MoveJ RelTool (starting_position, 116, -300, -124 \Rx:=7.8, \Ry:=-3, \Rz:=0), v200, z200, Tooldata_7;
MoveJ RelTool (starting_position, 117, -300, -124 \Rx:=7.6, \Ry:=-3, \Rz:=0), v200, z200, Tooldata_7;
MoveJ RelTool (starting_position, 117, -300, -124 \Rx:=7.4, \Ry:=-3, \Rz:=0), v200, z200, Tooldata_7;
MoveJ RelTool (starting_position, 117, -300, -123 \Rx:=7.2, \Ry:=-3, \Rz:=0), v200, z200, Tooldata_7;
MoveJ RelTool (starting_position, 118, -300, -123 \Rx:=6.9, \Ry:=-2.7, \Rz:=0), v200, z200, Tooldata_7;
MoveJ RelTool (starting_position, 118, -300, -123 \Rx:=6.6, \Ry:=-2.7, \Rz:=0), v200, z200, Tooldata_7;
MoveJ RelTool (starting_position, 119, -300, -122 \Rx:=6.2, \Ry:=-2.7, \Rz:=0), v200, z200, Tooldata_7;
MoveJ RelTool (starting_position, 119, -300, -122 \Rx:=5.8, \Ry:=-2.4, \Rz:=0), v200, z200, Tooldata_7;
MoveJ RelTool (starting_position, 120, -300, -122 \Rx:=5.4, \Ry:=-2.4, \Rz:=0), v200, z200, Tooldata_7;
MoveJ RelTool (starting_position, 120, -300, -121 \Rx:=4.9, \Ry:=-2.4, \Rz:=0), v200, z200, Tooldata_7;
MoveJ RelTool (starting_position, 121, -300, -121 \Rx:=4.4, \Ry:=-2.1, \Rz:=0), v200, z200, Tooldata_7;
MoveJ RelTool (starting_position, 121, -300, -121 \Rx:=3.9, \Ry:=-2.1, \Rz:=0), v200, z200, Tooldata_7;
MoveJ RelTool (starting_position, 122, -300, -120 \Rx:=3.5, \Ry:=-2.1, \Rz:=0), v200, z200, Tooldata_7;
MoveJ RelTool (starting_position, 123, -300, -120 \Rx:=3, \Ry:=-2.1, \Rz:=0), v200, z200, Tooldata_7;
MoveJ RelTool (starting_position, 124, -300, -119 \Rx:=2.6, \Ry:=-1.8, \Rz:=0), v200, z200, Tooldata_7;
MoveJ RelTool (starting_position, 125, -300, -119 \Rx:=2.2, \Ry:=-1.5, \Rz:=0), v200, z200, Tooldata_7;
MoveJ RelTool (starting_position, 126, -300, -119 \Rx:=1.7, \Ry:=-1.2, \Rz:=0), v200, z200, Tooldata_7;
MoveJ RelTool (starting_position, 127, -300, -119 \Rx:=1.3, \Ry:=-1.2, \Rz:=0), v200, z200, Tooldata_7;
MoveJ RelTool (starting_position, 127, -300, -118 \Rx:=0.9, \Ry:=-1.2, \Rz:=0), v200, z200, Tooldata_7;
MoveJ RelTool (starting_position, 128, -300, -118 \Rx:=0.5, \Ry:=-0.9, \Rz:=0), v200, z200, Tooldata_7;
MoveJ RelTool (starting_position, 129, -300, -118 \Rx:=0.2, \Ry:=-0.9, \Rz:=0), v200, z200, Tooldata_7;
MoveJ RelTool (starting_position, 130, -300, -118 \Rx:=-0.2, \Ry:=-0.6, \Rz:=0), v200, z200, Tooldata_7;
MoveJ RelTool (starting_position, 131, -300, -118 \Rx:=-0.5, \Ry:=-0.6, \Rz:=0), v200, z200, Tooldata_7;
MoveJ RelTool (starting_position, 132, -300, -118 \Rx:=-0.8, \Ry:=-0.3, \Rz:=0), v200, z200, Tooldata_7;
MoveJ RelTool (starting_position, 133, -300, -118 \Rx:=-1, \Ry:=-0, \Rz:=0), v200, z200, Tooldata_7;
MoveJ RelTool (starting_position, 134, -300, -118 \Rx:=-1.3, \Ry:=0, \Rz:=0), v200, z200, Tooldata_7;
MoveJ RelTool (starting_position, 135, -300, -118 \Rx:=-1.5, \Ry:=0.3, \Rz:=0), v200, z200, Tooldata_7;
MoveJ RelTool (starting_position, 136, -300, -118 \Rx:=-1.7, \Ry:=0.3, \Rz:=0), v200, z200, Tooldata_7;
MoveJ RelTool (starting_position, 137, -300, -118 \Rx:=-1.8, \Ry:=0.6, \Rz:=0), v200, z200, Tooldata_7;
MoveJ RelTool (starting_position, 138, -300, -118 \Rx:=-2, \Ry:=0.6, \Rz:=0), v200, z200, Tooldata_7;
MoveJ RelTool (starting_position, 139, -300, -119 \Rx:=-2, \Ry:=0.9, \Rz:=0), v200, z200, Tooldata_7;
MoveJ RelTool (starting_position, 140, -300, -119 \Rx:=-2.1, \Ry:=1.2, \Rz:=0), v200, z200, Tooldata_7;
MoveJ RelTool (starting_position, 141, -300, -119 \Rx:=-2.2, \Ry:=1.2, \Rz:=0), v200, z200, Tooldata_7;
MoveJ RelTool (starting_position, 142, -300, -119 \Rx:=-2.1, \Ry:=1.5, \Rz:=0), v200, z200, Tooldata_7;
MoveJ RelTool (starting_position, 142, -300, -120 \Rx:=-2.1, \Ry:=1.5, \Rz:=0), v200, z200, Tooldata_7;
MoveJ RelTool (starting_position, 143, -300, -120 \Rx:=-2, \Ry:=1.5, \Rz:=0), v200, z200, Tooldata_7;
MoveJ RelTool (starting_position, 144, -300, -120 \Rx:=-1.9, \Ry:=1.8, \Rz:=0), v200, z200, Tooldata_7;
MoveJ RelTool (starting_position, 145, -300, -121 \Rx:=-1.8, \Ry:=1.8, \Rz:=0), v200, z200, Tooldata_7;
MoveJ RelTool (starting_position, 145, -300, -121 \Rx:=-1.7, \Ry:=2.1, \Rz:=0), v200, z200, Tooldata_7;
MoveJ RelTool (starting_position, 146, -300, -121 \Rx:=-1.5, \Ry:=2.1, \Rz:=0), v200, z200, Tooldata_7;
MoveJ RelTool (starting_position, 147, -300, -122 \Rx:=-1.3, \Ry:=2.4, \Rz:=0), v200, z200, Tooldata_7;
MoveJ RelTool (starting_position, 148, -300, -122 \Rx:=-1.2, \Ry:=2.4, \Rz:=0), v200, z200, Tooldata_7;
MoveJ RelTool (starting_position, 148, -300, -122 \Rx:=-1, \Ry:=2.4, \Rz:=0), v200, z200, Tooldata_7;
MoveJ RelTool (starting_position, 149, -300, -123 \Rx:=-0.8, \Ry:=2.7, \Rz:=0), v200, z200, Tooldata_7;
MoveJ RelTool (starting_position, 149, -300, -123 \Rx:=-0.6, \Ry:=2.7, \Rz:=0), v200, z200, Tooldata_7;
MoveJ RelTool (starting_position, 150, -300, -123 \Rx:=-0.5, \Ry:=2.7, \Rz:=0), v200, z200, Tooldata_7;
MoveJ RelTool (starting_position, 150, -300, -123 \Rx:=-0.2, \Ry:=2.7, \Rz:=0), v200, z200, Tooldata_7;
MoveJ RelTool (starting_position, 151, -300, -124 \Rx:=-0, \Ry:=3, \Rz:=0), v200, z200, Tooldata_7;
MoveJ RelTool (starting_position, 151, -300, -124 \Rx:=0.1, \Ry:=3, \Rz:=0), v200, z200, Tooldata_7;
MoveJ RelTool (starting_position, 152, -300, -124 \Rx:=0.4, \Ry:=3.3, \Rz:=0), v200, z200, Tooldata_7;
MoveJ RelTool (starting_position, 153, -300, -124 \Rx:=0.6, \Ry:=3.3, \Rz:=0), v200, z200, Tooldata_7;
MoveJ RelTool (starting_position, 153, -300, -124 \Rx:=0.8, \Ry:=3.3, \Rz:=0), v200, z200, Tooldata_7;
MoveJ RelTool (starting_position, 154, -300, -125 \Rx:=1, \Ry:=3.6, \Rz:=0), v200, z200, Tooldata_7;
MoveJ RelTool (starting_position, 154, -300, -125 \Rx:=1.2, \Ry:=3.6, \Rz:=0), v200, z200, Tooldata_7;
MoveJ RelTool (starting_position, 155, -300, -125 \Rx:=1.5, \Ry:=3.6, \Rz:=0), v200, z200, Tooldata_7;
MoveJ RelTool (starting_position, 155, -300, -126 \Rx:=1.7, \Ry:=3.6, \Rz:=0), v200, z200, Tooldata_7;
MoveJ RelTool (starting_position, 156, -300, -126 \Rx:=1.9, \Ry:=3.9, \Rz:=0), v200, z200, Tooldata_7;
MoveJ RelTool (starting_position, 156, -300, -126 \Rx:=2.1, \Ry:=3.9, \Rz:=0), v200, z200, Tooldata_7;
MoveJ RelTool (starting_position, 157, -300, -127 \Rx:=2.3, \Ry:=3.9, \Rz:=0), v200, z200, Tooldata_7;
MoveJ RelTool (starting_position, 158, -300, -127 \Rx:=2.5, \Ry:=4.2, \Rz:=0), v200, z200, Tooldata_7;
MoveJ RelTool (starting_position, 158, -300, -128 \Rx:=2.7, \Ry:=4.2, \Rz:=0), v200, z200, Tooldata_7;
MoveJ RelTool (starting_position, 159, -300, -128 \Rx:=2.9, \Ry:=4.5, \Rz:=0), v200, z200, Tooldata_7;
MoveJ RelTool (starting_position, 160, -300, -128 \Rx:=3, \Ry:=4.5, \Rz:=0), v200, z200, Tooldata_7;
MoveJ RelTool (starting_position, 160, -300, -129 \Rx:=3.1, \Ry:=4.5, \Rz:=0), v200, z200, Tooldata_7;
MoveJ RelTool (starting_position, 161, -300, -129 \Rx:=3.2, \Ry:=4.8, \Rz:=0), v200, z200, Tooldata_7;
MoveJ RelTool (starting_position, 161, -300, -130 \Rx:=3.3, \Ry:=4.8, \Rz:=0), v200, z200, Tooldata_7;
MoveJ RelTool (starting_position, 162, -300, -131 \Rx:=3.3, \Ry:=4.8, \Rz:=0), v200, z200, Tooldata_7;
MoveJ RelTool (starting_position, 162, -300, -131 \Rx:=3.4, \Ry:=4.8, \Rz:=0), v200, z200, Tooldata_7;
MoveJ RelTool (starting_position, 162, -300, -132 \Rx:=3.4, \Ry:=5.1, \Rz:=0), v200, z200, Tooldata_7;
MoveJ RelTool (starting_position, 163, -300, -132 \Rx:=3.4, \Ry:=5.1, \Rz:=0), v200, z200, Tooldata_7;
MoveJ RelTool (starting_position, 163, -300, -133 \Rx:=3.4, \Ry:=5.1, \Rz:=0), v200, z200, Tooldata_7;
MoveJ RelTool (starting_position, 163, -300, -134 \Rx:=3.4, \Ry:=5.1, \Rz:=0), v200, z200, Tooldata_7;
MoveJ RelTool (starting_position, 163, -300, -134 \Rx:=3.3, \Ry:=5.1, \Rz:=0), v200, z200, Tooldata_7;
MoveJ RelTool (starting_position, 163, -300, -135 \Rx:=3.2, \Ry:=5.1, \Rz:=0), v200, z200, Tooldata_7;
MoveJ RelTool (starting_position, 163, -300, -135 \Rx:=3.1, \Ry:=5.1, \Rz:=0), v200, z200, Tooldata_7;
MoveJ RelTool (starting_position, 163, -300, -136 \Rx:=3, \Ry:=5.1, \Rz:=0), v200, z200, Tooldata_7;
MoveJ RelTool (starting_position, 163, -300, -136 \Rx:=2.9, \Ry:=5.1, \Rz:=0), v200, z200, Tooldata_7;
MoveJ RelTool (starting_position, 164, -300, -137 \Rx:=2.8, \Ry:=5.1, \Rz:=0), v200, z200, Tooldata_7;
MoveJ RelTool (starting_position, 164, -300, -138 \Rx:=2.7, \Ry:=5.1, \Rz:=0), v200, z200, Tooldata_7;
MoveJ RelTool (starting_position, 164, -300, -138 \Rx:=2.5, \Ry:=5.4, \Rz:=0), v200, z200, Tooldata_7;
MoveJ RelTool (starting_position, 165, -300, -139 \Rx:=2.4, \Ry:=5.4, \Rz:=0), v200, z200, Tooldata_7;
MoveJ RelTool (starting_position, 165, -300, -139 \Rx:=2.4, \Ry:=5.4, \Rz:=0), v200, z200, Tooldata_7;
MoveJ RelTool (starting_position, 165, -300, -140 \Rx:=2.4, \Ry:=5.4, \Rz:=0), v200, z200, Tooldata_7;
MoveJ RelTool (starting_position, 165, -300, -140 \Rx:=2.2, \Ry:=5.4, \Rz:=0), v200, z200, Tooldata_7;
MoveJ RelTool (starting_position, 165, -300, -141 \Rx:=2.1, \Ry:=5.4, \Rz:=0), v200, z200, Tooldata_7;
MoveJ RelTool (starting_position, 165, -300, -141 \Rx:=1.9, \Ry:=5.4, \Rz:=0), v200, z200, Tooldata_7;
MoveJ RelTool (starting_position, 165, -300, -142 \Rx:=1.9, \Ry:=5.4, \Rz:=0), v200, z200, Tooldata_7;
MoveJ RelTool (starting_position, 165, -300, -142 \Rx:=1.9, \Ry:=5.4, \Rz:=0), v200, z200, Tooldata_7;
MoveJ RelTool (starting_position, 165, -300, -143 \Rx:=1.9, \Ry:=5.7, \Rz:=0), v200, z200, Tooldata_7;
MoveJ RelTool (starting_position, 165, -300, -143 \Rx:=1.8, \Ry:=5.4, \Rz:=0), v200, z200, Tooldata_7;
MoveJ RelTool (starting_position, 165, -300, -144 \Rx:=1.8, \Ry:=5.4, \Rz:=0), v200, z200, Tooldata_7;
MoveJ RelTool (starting_position, 165, -300, -144 \Rx:=1.8, \Ry:=5.4, \Rz:=0), v200, z200, Tooldata_7;
MoveJ RelTool (starting_position, 165, -300, -145 \Rx:=1.8, \Ry:=5.4, \Rz:=0), v200, z200, Tooldata_7;
MoveJ RelTool (starting_position, 165, -300, -145 \Rx:=1.8, \Ry:=5.4, \Rz:=0), v200, z200, Tooldata_7;
MoveJ RelTool (starting_position, 165, -300, -146 \Rx:=1.8, \Ry:=5.4, \Rz:=0), v200, z200, Tooldata_7;
MoveJ RelTool (starting_position, 165, -300, -146 \Rx:=1.8, \Ry:=5.4, \Rz:=0), v200, z200, Tooldata_7;
MoveJ RelTool (starting_position, 165, -300, -147 \Rx:=1.8, \Ry:=5.4, \Rz:=0), v200, z200, Tooldata_7;
MoveJ RelTool (starting_position, 165, -300, -148 \Rx:=1.7, \Ry:=5.4, \Rz:=0), v200, z200, Tooldata_7;
MoveJ RelTool (starting_position, 165, -300, -148 \Rx:=1.7, \Ry:=5.4, \Rz:=0), v200, z200, Tooldata_7;
MoveJ RelTool (starting_position, 165, -300, -149 \Rx:=1.6, \Ry:=5.4, \Rz:=0), v200, z200, Tooldata_7;
MoveJ RelTool (starting_position, 165, -300, -149 \Rx:=1.6, \Ry:=5.4, \Rz:=0), v200, z200, Tooldata_7;
MoveJ RelTool (starting_position, 165, -300, -150 \Rx:=1.5, \Ry:=5.4, \Rz:=0), v200, z200, Tooldata_7;
MoveJ RelTool (starting_position, 165, -300, -151 \Rx:=1.4, \Ry:=5.4, \Rz:=0), v200, z200, Tooldata_7;
MoveJ RelTool (starting_position, 165, -300, -151 \Rx:=1.2, \Ry:=5.4, \Rz:=0), v200, z200, Tooldata_7;
MoveJ RelTool (starting_position, 165, -300, -152 \Rx:=1.1, \Ry:=5.4, \Rz:=0), v200, z200, Tooldata_7;
MoveJ RelTool (starting_position, 165, -300, -153 \Rx:=1, \Ry:=5.4, \Rz:=0), v200, z200, Tooldata_7;
MoveJ RelTool (starting_position, 165, -300, -153 \Rx:=0.9, \Ry:=5.4, \Rz:=0), v200, z200, Tooldata_7;
MoveJ RelTool (starting_position, 165, -300, -154 \Rx:=0.8, \Ry:=5.4, \Rz:=0), v200, z200, Tooldata_7;
MoveJ RelTool (starting_position, 164, -300, -154 \Rx:=0.6, \Ry:=5.4, \Rz:=0), v200, z200, Tooldata_7;
MoveJ RelTool (starting_position, 164, -300, -155 \Rx:=0.5, \Ry:=5.1, \Rz:=0), v200, z200, Tooldata_7;
MoveJ RelTool (starting_position, 164, -300, -155 \Rx:=0.4, \Ry:=5.1, \Rz:=0), v200, z200, Tooldata_7;
MoveJ RelTool (starting_position, 163, -300, -156 \Rx:=0.2, \Ry:=5.1, \Rz:=0), v200, z200, Tooldata_7;
MoveJ RelTool (starting_position, 163, -300, -156 \Rx:=0.1, \Ry:=5.1, \Rz:=0), v200, z200, Tooldata_7;
MoveJ RelTool (starting_position, 163, -300, -157 \Rx:=-0, \Ry:=5.1, \Rz:=0), v200, z200, Tooldata_7;
MoveJ RelTool (starting_position, 163, -300, -157 \Rx:=-0.1, \Ry:=5.1, \Rz:=0), v200, z200, Tooldata_7;
MoveJ RelTool (starting_position, 162, -300, -158 \Rx:=-0.2, \Ry:=5.1, \Rz:=0), v200, z200, Tooldata_7;
MoveJ RelTool (starting_position, 162, -300, -158 \Rx:=-0.3, \Ry:=4.8, \Rz:=0), v200, z200, Tooldata_7;
MoveJ RelTool (starting_position, 162, -300, -159 \Rx:=-0.4, \Ry:=4.8, \Rz:=0), v200, z200, Tooldata_7;
MoveJ RelTool (starting_position, 162, -300, -159 \Rx:=-0.5, \Ry:=4.8, \Rz:=0), v200, z200, Tooldata_7;
MoveJ RelTool (starting_position, 161, -300, -160 \Rx:=-0.6, \Ry:=4.8, \Rz:=0), v200, z200, Tooldata_7;
MoveJ RelTool (starting_position, 161, -300, -160 \Rx:=-0.7, \Ry:=4.8, \Rz:=0), v200, z200, Tooldata_7;
MoveJ RelTool (starting_position, 161, -300, -161 \Rx:=-0.8, \Ry:=4.8, \Rz:=0), v200, z200, Tooldata_7;
MoveJ RelTool (starting_position, 160, -300, -161 \Rx:=-0.9, \Ry:=4.5, \Rz:=0), v200, z200, Tooldata_7;
MoveJ RelTool (starting_position, 160, -300, -162 \Rx:=-0.9, \Ry:=4.5, \Rz:=0), v200, z200, Tooldata_7;
MoveJ RelTool (starting_position, 160, -300, -162 \Rx:=-1, \Ry:=4.5, \Rz:=0), v200, z200, Tooldata_7;
MoveJ RelTool (starting_position, 160, -300, -162 \Rx:=-1.1, \Ry:=4.5, \Rz:=0), v200, z200, Tooldata_7;
MoveJ RelTool (starting_position, 159, -300, -163 \Rx:=-1.1, \Ry:=4.5, \Rz:=0), v200, z200, Tooldata_7;
MoveJ RelTool (starting_position, 159, -300, -163 \Rx:=-1.1, \Ry:=4.5, \Rz:=0), v200, z200, Tooldata_7;
MoveJ RelTool (starting_position, 159, -300, -164 \Rx:=-1.2, \Ry:=4.2, \Rz:=0), v200, z200, Tooldata_7;
MoveJ RelTool (starting_position, 158, -300, -164 \Rx:=-1.2, \Ry:=4.2, \Rz:=0), v200, z200, Tooldata_7;
MoveJ RelTool (starting_position, 158, -300, -164 \Rx:=-1.2, \Ry:=4.2, \Rz:=0), v200, z200, Tooldata_7;
MoveJ RelTool (starting_position, 158, -300, -165 \Rx:=-1.3, \Ry:=4.2, \Rz:=0), v200, z200, Tooldata_7;
MoveJ RelTool (starting_position, 157, -300, -165 \Rx:=-1.4, \Ry:=4.2, \Rz:=0), v200, z200, Tooldata_7;
MoveJ RelTool (starting_position, 157, -300, -165 \Rx:=-1.3, \Ry:=3.9, \Rz:=0), v200, z200, Tooldata_7;
MoveJ RelTool (starting_position, 157, -300, -166 \Rx:=-1.3, \Ry:=3.9, \Rz:=0), v200, z200, Tooldata_7;























        !MoveJ [ [0, 0, 1225], [-0.282, 0.072, 0.956, 0.021], [0, -1,-1, 1], [0, 9E9, 9E9, 9E9, 9E9, 9E9] ],v20,z1,Tooldata_7;
        !MoveJ [ [0, 0, 1000], [-0.282, 0.072, 0.956, 0.021], [0, -1,-1, 1], [0, 9E9, 9E9, 9E9, 9E9, 9E9] ],v20,z1,Tooldata_7;
        !EGM_CARTESIAN_MOVE;
       ! RAPID_MOVE;

    ENDPROC

    ! ################################## Externally Guided motion (EGM) - Cartesian Control ################################## !



ENDMODULE
